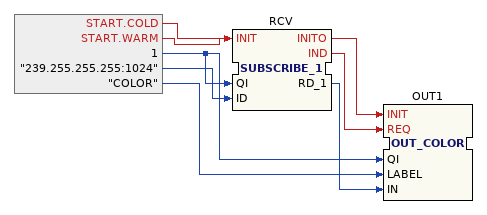
      FBS
        RCV : SUBSCRIBE_1;
        OUT1 : OUT_COLOR;
      END_FBS
      EVENT_CONNECTIONS
        START.COLD TO RCV.INIT;
        START.WARM TO RCV.INIT;
        RCV.INITO TO OUT1.INIT;
        RCV.IND TO OUT1.REQ;
      END_CONNECTIONS
      DATA_CONNECTIONS
        1 TO RCV.QI;
        "239.255.255.255:1024" TO RCV.ID;
        1 TO OUT1.QI;
        "COLOR" TO OUT1.LABEL;
        RCV.RD_1 TO OUT1.IN;
      END_CONNECTIONS
    END_RESOURCE
    DATA_CONNECTIONS
      0 TO RES0.TRACE;
    END_CONNECTIONS
  END_DEVICE
  DATA_CONNECTIONS (* parameter values *)
    [50,50,175,195] TO SEND_BITS.BOUNDS;
    [225,50,175,195] TO RCV_BITS.BOUNDS;
    [50,240,175,170] TO SEND_INTS.BOUNDS;
    [225,240,175,170] TO RCV_INTS.BOUNDS;
    [50,405,175,120] TO SEND_UINTS.BOUNDS;
    [225,405,175,120] TO RCV_UINTS.BOUNDS;
    [50,520,175,90] TO SEND_REALS.BOUNDS;
    [225,520,175,90] TO RCV_REALS.BOUNDS;
    [400,50,400,225] TO MONITOR.BOUNDS;
    [400,270,200,115] TO SEND_TIMES.BOUNDS;
    [600,270,200,115] TO RCV_TIMES.BOUNDS;
    [400,385,200,95] TO SEND_STRINGS.BOUNDS;
    [600,385,200,95] TO RCV_STRINGS.BOUNDS;
    [400,480,210,65] TO SEND_ARRAY.BOUNDS;
    [610,480,190,65] TO RCV_ARRAY.BOUNDS;
    [400,540,210,70] TO SEND_COLOR.BOUNDS;
    [610,540,190,70] TO RCV_COLOR.BOUNDS;
    [1,1] TO SEND_BITS.GRID;
    [1,1] TO RCV_BITS.GRID;
    [1,1] TO SEND_INTS.GRID;
    [1,1] TO RCV_INTS.GRID;
    [1,1] TO SEND_UINTS.GRID;
    [1,1] TO RCV_UINTS.GRID;
    [1,1] TO SEND_REALS.GRID;
    [1,1] TO RCV_REALS.GRID;
    [1,1] TO SEND_TIMES.GRID;
    [1,1] TO RCV_TIMES.GRID;
    [1,1] TO SEND_STRINGS.GRID;
    [1,1] TO RCV_STRINGS.GRID;
    [1,1] TO SEND_ARRAY.GRID;
    [1,1] TO RCV_ARRAY.GRID;
    [1,1] TO SEND_COLOR.GRID;
    [1,1] TO RCV_COLOR.GRID;
    [1,1] TO MONITOR.GRID;
  END_CONNECTIONS
  MAPPINGS
    TEST_BITS.IN0 ON SEND_BITS.RES0.IN0;
    TEST_BITS.OUT0 ON RCV_BITS.RES0.OUT0;
    TEST_BITS.IN1 ON SEND_BITS.RES0.IN1;
    TEST_BITS.OUT1 ON RCV_BITS.RES0.OUT1;
    TEST_BITS.PB21 ON SEND_BITS.RES0.PB21;
    TEST_BITS.IN21 ON SEND_BITS.RES0.IN21;
    TEST_BITS.PB22 ON SEND_BITS.RES0.PB22;
    TEST_BITS.OUT21 ON RCV_BITS.RES0.OUT21;
    TEST_BITS.IN22 ON SEND_BITS.RES0.IN22;
    TEST_BITS.OUT22 ON RCV_BITS.RES0.OUT22;
    TEST_BITS.PB31 ON SEND_BITS.RES0.PB31;
    TEST_BITS.IN31 ON SEND_BITS.RES0.IN31;
    TEST_BITS.OUT31 ON RCV_BITS.RES0.OUT31;
    TEST_BITS.PB32 ON SEND_BITS.RES0.PB32;
    TEST_BITS.IN32 ON SEND_BITS.RES0.IN32;
    TEST_BITS.OUT32 ON RCV_BITS.RES0.OUT32;
    TEST_INTS.PB1 ON SEND_INTS.RES0.PB1;
    TEST_INTS.IN1 ON SEND_INTS.RES0.IN1;
    TEST_INTS.PB2 ON SEND_INTS.RES0.PB2;
    TEST_INTS.IN2 ON SEND_INTS.RES0.IN2;
    TEST_INTS.PB3 ON SEND_INTS.RES0.PB3;
    TEST_INTS.IN3 ON SEND_INTS.RES0.IN3;
    TEST_INTS.PB4 ON SEND_INTS.RES0.PB4;
    TEST_INTS.IN4 ON SEND_INTS.RES0.IN4;
    TEST_INTS.OUT1 ON RCV_INTS.RES0.OUT1;
    TEST_INTS.OUT2 ON RCV_INTS.RES0.OUT2;
    TEST_INTS.OUT3 ON RCV_INTS.RES0.OUT3;
    TEST_INTS.OUT4 ON RCV_INTS.RES0.OUT4;
    TEST_UINTS.PB1 ON SEND_UINTS.RES0.PB1;
    TEST_UINTS.IN1 ON SEND_UINTS.RES0.IN1;
    TEST_UINTS.PB2 ON SEND_UINTS.RES0.PB2;
    TEST_UINTS.IN2 ON SEND_UINTS.RES0.IN2;
    TEST_UINTS.PB3 ON SEND_UINTS.RES0.PB3;
    TEST_UINTS.IN3 ON SEND_UINTS.RES0.IN3;
    TEST_UINTS.OUT1 ON RCV_UINTS.RES0.OUT1;
    TEST_UINTS.OUT2 ON RCV_UINTS.RES0.OUT2;
    TEST_UINTS.OUT3 ON RCV_UINTS.RES0.OUT3;
    TEST_REALS.PB1 ON SEND_REALS.RES0.PB1;
    TEST_REALS.IN1 ON SEND_REALS.RES0.IN1;
    TEST_REALS.PB2 ON SEND_REALS.RES0.PB2;
    TEST_REALS.IN2 ON SEND_REALS.RES0.IN2;
    TEST_REALS.OUT1 ON RCV_REALS.RES0.OUT1;
    TEST_REALS.OUT2 ON RCV_REALS.RES0.OUT2;
    TEST_TIMES.PB1 ON SEND_TIMES.RES0.PB1;
    TEST_TIMES.IN1 ON SEND_TIMES.RES0.IN1;
    TEST_TIMES.PB2 ON SEND_TIMES.RES0.PB2;
    TEST_TIMES.IN2 ON SEND_TIMES.RES0.IN2;
    TEST_TIMES.OUT1 ON RCV_TIMES.RES0.OUT1;
    TEST_TIMES.OUT2 ON RCV_TIMES.RES0.OUT2;
    TEST_STRINGS.PB1 ON SEND_STRINGS.RES0.PB1;
    TEST_STRINGS.IN1 ON SEND_STRINGS.RES0.IN1;
    TEST_STRINGS.PB2 ON SEND_STRINGS.RES0.PB2;
    TEST_STRINGS.IN2 ON SEND_STRINGS.RES0.IN2;
    TEST_STRINGS.OUT1 ON RCV_STRINGS.RES0.OUT1;
    TEST_STRINGS.OUT2 ON RCV_STRINGS.RES0.OUT2;
    TEST_ARRAY.PB1 ON SEND_ARRAY.RES0.PB1;
    TEST_ARRAY.IN1 ON SEND_ARRAY.RES0.PB1;
    TEST_ARRAY.OUT1 ON RCV_ARRAY.RES0.OUT1;
    TEST_COLOR.IN1 ON SEND_COLOR.RES0.IN1;
    TEST_COLOR.OUT1 ON RCV_COLOR.RES0.OUT1;
  END_MAPPINGS
END_SYSTEM
